FUNCTION_BLOCK ReflectionTest EXTENDS TcUnit.FB_TestSuite
VAR
	reflection : Reflection(THIS, SIZEOF(THIS^));
END_VAR

GetAllData();

METHOD GetAllData : BOOL
VAR
END_VAR
TcUnit.TEST('Get all data');

AssertEquals_STRING(
	Actual := reflection.InstanceName,
	Expected := 'FrameworkMonorepoTests.FMTypesTests.PRG_Test.reflectionTest',
	Message := 'InstanceName was not obtained correctly');

AssertEquals_STRING(
	Actual := reflection.SolutionName,
	Expected := 'FrameworkMonorepoTests',
	Message := 'SolutionName was not obtained correctly');

AssertEquals_STRING(
	Actual := reflection.ProjectName,
	Expected := 'FMTypesTests',
	Message := 'ProjectName was not obtained correctly');

AssertEquals_STRING(
	Actual := reflection.ParentName,
	Expected := 'PRG_Test',
	Message := 'ParentName was not obtained correctly');

AssertEquals_STRING(
	Actual := reflection.Name,
	Expected := 'reflectionTest',
	Message := 'Name was not obtained correctly');

AssertEquals_STRING(
	Actual := reflection.ObjectPath,
	Expected := 'PRG_Test.reflectionTest',
	Message := 'ObjectPath was not obtained correctly');

AssertEquals_STRING(
	Actual := reflection.TypeName,
	Expected := 'ReflectionTest',
	Message := 'TypeName was not obtained correctly');

TEST_FINISHED();
END_METHOD

END_FUNCTION_BLOCK

(* stored: Version 1.1.0.1, ProductVersion 3.1.4024.15
   POU ReflectionTest: Id {f12a370c-bcbc-088d-3cc3-c89575cfef88}, SpecialFunc None
   Method GetAllData: Id {9926ef1f-d076-0efd-3a93-f80c25b9ed12} *)
